// TIA Portal V17 export
// export: Created 2024-09-02T12:50:36.1664401Z, ExportSetting WithDefaults, DisplayName Totally Integrated Automation Portal, DisplayVersion V17, DisplayName TIA Portal Openness, DisplayVersion V17, DisplayName TIA Portal Version Control Interface, DisplayVersion V17, DisplayName STEP 7 Professional, DisplayVersion V17, DisplayName STEP 7 Safety, DisplayVersion V17, DisplayName WinCC Professional, DisplayVersion V17
TYPE "TypeMobyKEY_1"
// stored: IsFailsafeCompliant false
   STRUCT
      KST_1 : Char;   // Kostenstelle / Cost centre
      KST_2 : Char;   // Kostenstelle / Cost centre
      KST_3 : Char;   // Kostenstelle / Cost centre
      KST_4 : Char;   // Kostenstelle / Cost centre
      MA_NR_1 : Char;   // Mitarbeiter / Employees
      MA_NR_2 : Char;   // Mitarbeiter / Employees
      MA_NR_3 : Char;   // Mitarbeiter / Employees
      MA_NR_4 : Char;   // Mitarbeiter / Employees
      STUFE : Char;   // Berechtigung / Permission
      JAHR : Byte;   // Zeitstempel / Time stamp
      MONAT : Byte;   // Zeitstempel / Time stamp
      TAG : Byte;   // Zeitstempel / Time stamp
      STUNDE : Byte;   // Zeitstempel / Time stamp
      MINUTE : Byte;   // Zeitstempel / Time stamp
      SEKUNDE : Byte;   // Zeitstempel / Time stamp
      ERST_KST_1 : Char;   // Kostenstelle - Erstwert / Cost center - initial value
      ERST_KST_2 : Char;   // Kostenstelle - Erstwert / Cost center - initial value
      ERST_KST_3 : Char;   // Kostenstelle - Erstwert / Cost center - initial value
      ERST_KST_4 : Char;   // Kostenstelle - Erstwert / Cost center - initial value
      ERST_MA_NR_1 : Char;   // Mitarbeiter - Erstwert / Employees - first value
      ERST_MA_NR_2 : Char;   // Mitarbeiter - Erstwert / Employees - first value
      ERST_MA_NR_3 : Char;   // Mitarbeiter - Erstwert / Employees - first value
      ERST_MA_NR_4 : Char;   // Mitarbeiter - Erstwert / Employees - first value
      ERST_STUFE : Char;   // Berechtigung - Erstwert / Permission - First value
      ERST_JAHR : Byte;   // Zeitstempel - Erstwert / Timestamp - First value
      ERST_MONAT : Byte;   // Zeitstempel - Erstwert / Timestamp - First value
      ERST_TAG : Byte;   // Zeitstempel - Erstwert / Timestamp - First value
      ERST_STUNDE : Byte;   // Zeitstempel - Erstwert / Timestamp - First value
      ERST_MINUTE : Byte;   // Zeitstempel - Erstwert / Timestamp - First value
      ERST_SEKUNDE : Byte;   // Zeitstempel - Erstwert / Timestamp - First value
   END_STRUCT;
END_TYPE
